INTERFACE I_EM_LiftingTransport

END_INTERFACE

(* stored: Version 1.1.0.1, ProductVersion 3.1.4024.12
   Itf I_EM_LiftingTransport: Id {2a02f975-5ee0-48c3-ac02-e06ca2637228} *)
